(* PLC project  *)

CONFIGURATION Empty_Module_5
END_CONFIGURATION
